TYPE csp_transfer_accumulator_accU_virtualMaster_enum :
(
	CSP_TRANSFER_ACCUMULATOR_ACCU_VIRTUAL_MASTER_STATUS_NOT_INITIALIZED 								:= 0,
	CSP_TRANSFER_ACCUMULATOR_ACCU_VIRTUAL_MASTER_STATUS_DISABLED 										:= 10,
	CSP_TRANSFER_ACCUMULATOR_ACCU_VIRTUAL_MASTER_STATUS_POSITION_CHECK									:= 20,
	CSP_TRANSFER_ACCUMULATOR_ACCU_VIRTUAL_MASTER_STATUS_CHECK_SLAVE_GEAR 								:= 25,
	CSP_TRANSFER_ACCUMULATOR_ACCU_VIRTUAL_MASTER_STATUS_ENABLE_REQUEST 									:= 30,
	CSP_TRANSFER_ACCUMULATOR_ACCU_VIRTUAL_MASTER_STATUS_ENABLED 										:= 40,
	CSP_TRANSFER_ACCUMULATOR_ACCU_VIRTUAL_MASTER_STATUS_ABS_MOVE_REQUEST								:= 50,
	CSP_TRANSFER_ACCUMULATOR_ACCU_VIRTUAL_MASTER_STATUS_ABS_MOVING										:= 60,
	CSP_TRANSFER_ACCUMULATOR_ACCU_VIRTUAL_MASTER_STATUS_STOP_REQUEST 									:= 70,
	CSP_TRANSFER_ACCUMULATOR_ACCU_VIRTUAL_MASTER_STATUS_DISABLE_REQUEST 								:= 80,
	CSP_TRANSFER_ACCUMULATOR_ACCU_VIRTUAL_MASTER_STATUS_DISABLING 										:= 90
) := CSP_TRANSFER_ACCUMULATOR_ACCU_VIRTUAL_MASTER_STATUS_NOT_INITIALIZED;
END_TYPE

(* stored: Version 1.1.0.1, ProductVersion 3.1.4024.3
   DUT csp_transfer_accumulator_accU_virtualMaster_enum: Id {a13923b8-e7d1-479f-8d06-10f77a6aae08} *)
